FUNCTION_BLOCK Test_TExecutionWhenBusy_Start_RaisesNotification EXTENDS T_UnitTestbase
VAR
    Execution                            : T_Execution;
    ExecutionFailed_NotificationHandler  : T_NotificationHandler;
    ExecutionAborted_NotificationHandler : T_NotificationHandler;
END_VAR

METHOD Init
// Setup...
Execution.FB_init(bInitRetains := FALSE,
                  bInCopyCode  := FALSE);

ExecutionFailed_NotificationHandler.FB_init(bInitRetains := FALSE,
                                            bInCopyCode  := FALSE);

ExecutionAborted_NotificationHandler.FB_init(bInitRetains := FALSE,
                                             bInCopyCode  := FALSE);
END_METHOD

{attribute 'analysis' := '-33'} // inhibit unused variable warning
METHOD RunTest
VAR_OUTPUT
    TestCompleted : BOOL;
    TestFailed    : BOOL;
END_VAR
// link handler to common execution events...
GlobalNotifications.Notification_ExecutionFailed
    .ClearNotificationHandlers()
    .AddNotificationHandler(ExecutionFailed_NotificationHandler);

GlobalNotifications.Notification_ExecutionAborted
    .ClearNotificationHandlers()
    .AddNotificationHandler(ExecutionAborted_NotificationHandler);

// Test...
Execution.Start(); // sets Starting

Execution.Start(); // raises error event

TestFailed S= NOT AssertTrue(Source    := TestName,
                             Condition := ExecutionFailed_NotificationHandler.IsRaised(),
                             Message   := 'ExecutionFailed_NotificationHandler.IsRaised() not true');

TestCompleted := TRUE;
END_METHOD

END_FUNCTION_BLOCK

(* stored: Version 1.1.0.1, ProductVersion 3.1.4024.12
   POU Test_TExecutionWhenBusy_Start_RaisesNotification: Id {084b24e3-9990-483f-9341-dda52872d69c}, SpecialFunc None
   Method Init: Id {7b223d44-04c2-4411-99e7-7c0f85109818}
   Method RunTest: Id {0f92d60d-0ca0-44d2-8941-f0b332232631} *)
